// TIA Portal project "projeto_Grafcet" (V17)

(* hardware
DEVICE "S7-1500/ET200MP station_1"  S7-1500 station
   slot 0: "Rail_0"  Rack  6ES7 590-1***0-0AA0
   slot 1: "PLC_1"  CPU 1513-1 PN  6ES7 513-1AL02-0AB0  V2.9
      slot 3: "CPU display_1"  6ES7591-1AA00-0AA0
      slot 32768: "PROFINET interface_1"  X1
         slot 32769: "Port_1"  X1 P1
         slot 32770: "Port_2"  X1 P2
      slot 34817: "Virtual CP interface port_1"  Virtual CP interface port  Virtual CP interface port
   slot 2: "DI 32x24VDC SNK/SRC / DQ 32x24VDC/0.3A SNK BA_1"  DI 32x24VDC SNK/SRC / DQ 32x24VDC/0.3A SNK BA  6ES7 523-1BP50-0AA0  V1.0
*)

// ===== PLC "PLC_1"  CPU 1513-1 PN =====

VAR_GLOBAL   // PLC tag table "Default tag table"
   "Tag_3" AT %M2.2 : Bool;
   "Tag_4" AT %M2.0 : Bool;
   "Tag_1" AT %M2.4 : Bool;
   "Tag_5" AT %M2.5 : Bool;
   "Tag_2" AT %M3.3 : Bool;
   "Tag_6" AT %M3.4 : Bool;
   "Tag_7" AT %M2.6 : Bool;
   "Tag_8" AT %M2.7 : Bool;
   "Tag_9" AT %M3.0 : Bool;
   "Tag_10" AT %M3.1 : Bool;
   "M_1" AT %M1.3 : Bool;
   "M_2" AT %M1.4 : Bool;
   "MSaida" AT %M1.5 : Bool;
   "Limite Verde" AT %M1.6 : Bool;
   "MSAidaA" AT %M1.7 : Bool;
   "limite Azul" AT %M3.2 : Bool;
   "Mconta1" AT %M3.5 : Bool;
   "Mconta2" AT %M3.6 : Bool;
   "Terminou robo2" AT %M3.7 : Bool;
   "FACTORY I/O(Running)" AT %I1.7 : Bool;
   "Memo1" AT %M0.0 : Bool;
   "memo2" AT %M0.1 : Bool;
   "memo3" AT %M0.2 : Bool;
   "memo4" AT %M0.3 : Bool;
   "memo5" AT %M0.4 : Bool;
   "M_R2_Segura" AT %M0.5 : Bool;
   "M_R1_Segura" AT %M0.6 : Bool;
   "Limite_Ordenação" AT %M0.7 : Bool;
   "Sensor_borda_N" AT %M1.0 : Bool;
   "Fim_Etapa_Distribuição" AT %M1.1 : Bool;
   "termina_Distribuição" AT %M1.2 : Bool;
END_VAR

VAR_GLOBAL   // PLC tag table "Tag table_1"
   "R1 Sensor de Detecção de Peça" AT %I0.0 : Bool;
   "R2 Sensor de Detecção de Peça" AT %I0.1 : Bool;
   "R1 Sensor de Movimento Descer/Subir" AT %I0.2 : Bool;
   "R2 Sensor de Movimento Descer/Subir" AT %I0.3 : Bool;
   "R1 Sensor de Movimento Avançar/Recuar" AT %I0.4 : Bool;
   "R2 Sensor de Movimento Avançar/Recuar" AT %I0.5 : Bool;
   "Sensor de Saída 1" AT %I0.6 : Bool;
   "Sensor de Saída 2" AT %I0.7 : Bool;
   "Sensor do Organizador" AT %I1.0 : Bool;
   "Sensor Entrada Azul" AT %I1.1 : Bool;
   "Sensor Entrada Verde" AT %I1.2 : Bool;
   "Sensor Peça Azul" AT %I1.3 : Bool;
   "Sensor Peça Verde" AT %I1.4 : Bool;
   "Sensor Saída Azul" AT %I1.5 : Bool;
   "Sensor Saída Verde" AT %I1.6 : Bool;
   "Barreira" AT %Q0.0 : Bool;
   "Cinta do Desviador" AT %Q0.1 : Bool;
   "Deslocar Direita" AT %Q0.2 : Bool;
   "Deslocar Esquerda" AT %Q0.3 : Bool;
   "Desviador" AT %Q0.4 : Bool;
   "Esteira de Alimentação" AT %Q0.5 : Bool;
   "Esteira de Descarte P1" AT %Q0.6 : Bool;
   "Esteira de Descarte P2" AT %Q0.7 : Bool;
   "Esteira de Saída P1" AT %Q1.0 : Bool;
   "Esteira de Saída P2" AT %Q1.1 : Bool;
   "Esteira do Organizador" AT %Q1.2 : Bool;
   "Esteira Peça Azul  P1" AT %Q1.3 : Bool;
   "Esteira Peça Azul P2" AT %Q1.4 : Bool;
   "Esteira Peça Verde P1" AT %Q1.5 : Bool;
   "Esteira Peça Verde P2" AT %Q1.6 : Bool;
   "Esteira Peça Verde P3" AT %Q1.7 : Bool;
   "Esteira Peça Verde P4" AT %Q2.0 : Bool;
   "Esteira Peça Verde P5" AT %Q2.1 : Bool;
   "R1 Descer=1/Subir=0" AT %Q2.2 : Bool;
   "R2 Descer=1/Subir=0" AT %Q2.3 : Bool;
   "R1 Avançar=1/Recuar=0" AT %Q2.4 : Bool;
   "R1 Segurar=1/Soltar=0" AT %Q2.5 : Bool;
   "R2 Avançar=1/Recuar=0" AT %Q2.6 : Bool;
   "R2 Segurar=1/Soltar=0" AT %Q2.7 : Bool;
   "Receber Peça" AT %Q3.0 : Bool;
END_VAR

DATA_BLOCK "Separação_DB"   // DB6
{ S7_Optimized_Access := 'TRUE' }
VERSION : 0.1
// stored: InstanceOfName Separação
"Separação"
BEGIN
END_DATA_BLOCK

DATA_BLOCK "Block_1_DB"   // DB7
{ S7_Optimized_Access := 'TRUE' }
VERSION : 0.1
// stored: InstanceOfName Descarte
"Descarte"
BEGIN
END_DATA_BLOCK

DATA_BLOCK "Robo 2_DB"   // DB8
{ S7_Optimized_Access := 'TRUE' }
VERSION : 0.1
// stored: InstanceOfName Robo 2
"Robo 2"
BEGIN
END_DATA_BLOCK

DATA_BLOCK "Robo 1_DB"   // DB9
{ S7_Optimized_Access := 'TRUE' }
VERSION : 0.1
// stored: InstanceOfName Robo 1
"Robo 1"
BEGIN
END_DATA_BLOCK

DATA_BLOCK "Distribuição_DB"   // DB13
{ S7_Optimized_Access := 'TRUE' }
VERSION : 0.1
// stored: InstanceOfName Distribuição
"Distribuição"
BEGIN
END_DATA_BLOCK

// folder: System blocks/Program resources

DATA_BLOCK "IEC_Timer_0_DB"   // DB1
{ S7_Optimized_Access := 'TRUE' }
AUTHOR : Simatic
FAMILY : IEC
NAME : IEC_TMR
VERSION : 1.0
// stored: InstanceOfName IEC_TIMER
"IEC_TIMER"
BEGIN
END_DATA_BLOCK

DATA_BLOCK "IEC_Timer_0_DB_1"   // DB2
{ S7_Optimized_Access := 'TRUE' }
AUTHOR : Simatic
FAMILY : IEC
NAME : IEC_TMR
VERSION : 1.0
// stored: InstanceOfName IEC_TIMER
"IEC_TIMER"
BEGIN
END_DATA_BLOCK

DATA_BLOCK "IEC_Timer_0_DB_2"   // DB3
{ S7_Optimized_Access := 'TRUE' }
AUTHOR : Simatic
FAMILY : IEC
NAME : IEC_TMR
VERSION : 1.0
// stored: InstanceOfName IEC_TIMER
"IEC_TIMER"
BEGIN
END_DATA_BLOCK

DATA_BLOCK "IEC_Counter_0_DB"   // DB4
{ S7_Optimized_Access := 'TRUE' }
AUTHOR : Simatic
FAMILY : IEC
NAME : CNTR
VERSION : 1.0
// stored: InstanceOfName IEC_COUNTER
"IEC_COUNTER"
BEGIN
END_DATA_BLOCK

DATA_BLOCK "IEC_Counter_0_DB_1"   // DB5
{ S7_Optimized_Access := 'TRUE' }
AUTHOR : Simatic
FAMILY : IEC
NAME : CNTR
VERSION : 1.0
// stored: InstanceOfName IEC_COUNTER
"IEC_COUNTER"
BEGIN
END_DATA_BLOCK

DATA_BLOCK "IEC_Timer_0_DB_3"   // DB10
{ S7_Optimized_Access := 'TRUE' }
AUTHOR : Simatic
FAMILY : IEC
NAME : IEC_TMR
VERSION : 1.0
// stored: InstanceOfName IEC_TIMER
"IEC_TIMER"
BEGIN
END_DATA_BLOCK

DATA_BLOCK "IEC_Counter_0_DB_2"   // DB11
{ S7_Optimized_Access := 'TRUE' }
AUTHOR : Simatic
FAMILY : IEC
NAME : CNTR
VERSION : 1.0
// stored: InstanceOfName IEC_COUNTER
"IEC_COUNTER"
BEGIN
END_DATA_BLOCK

DATA_BLOCK "IEC_Counter_0_DB_3"   // DB12
{ S7_Optimized_Access := 'TRUE' }
AUTHOR : Simatic
FAMILY : IEC
NAME : CNTR
VERSION : 1.0
// stored: InstanceOfName IEC_COUNTER
"IEC_COUNTER"
BEGIN
END_DATA_BLOCK

// folder: (top level)

FUNCTION_BLOCK "Descarte"   // FB1, GRAPH_PLUS
{ S7_Optimized_Access := 'TRUE' }
VERSION : 0.1
   VAR_INPUT
      OFF_SQ : Bool := false;   // Turn sequence off
      INIT_SQ : Bool := false;   // Set sequence to initial state
      ACK_EF : Bool := false;   // Acknowledge all errors and faults
      S_PREV : Bool := false;   // Output previous step in parameter S_NO
      "Peça green" : Bool;
      S_NEXT : Bool := false;   // Indicate next step in parameter S_NO
      "peça blue" : Bool;
      SW_AUTO : Bool := false;   // Automatic mode
      SW_TAP : Bool := false;   // Semiautomatic/switch with transition
      SW_TOP : Bool := false;   // Semiautomatic/ignore transition
      SW_MAN : Bool := false;   // Manual mode
      S_SEL : Int := 0;   // Select step to be output to S_NO
      S_ON : Bool := false;   // Activate step indicated in S_NO
      S_OFF : Bool := false;   // Deactivate step indicated S_NO
      T_PUSH : Bool := false;   // Enable transition to switch in semi automatic mode
   END_VAR
   VAR_OUTPUT
      S_NO : Int := 0;   // Step number
      S_MORE : Bool := false;   // More steps are available and can be shown in S_NO
      S_ACTIVE : Bool := false;   // Step indicated in S_NO is active
      Cinta : Bool;
      ERR_FLT : Bool := false;   // Interlock or supervision group error
      AUTO_ON : Bool := false;   // Automatic mode is active
      D2 : Bool;
      D1 : Bool;
      Desviar_peça : Bool;
      TAP_ON : Bool := false;   // Semiautomatic mode/step with transition enabled
      TOP_ON : Bool := false;   // Semiautomatic mode/ignore transition enabled
      MAN_ON : Bool := false;   // Manual mode is active
   END_VAR
   VAR
      HMI_INFO : Array[0..8] of UInt;
      IF_PAR : G7_IfParPlus_V6;
      RT_DATA : G7_RTDataPlus_V6;   // Internal data area
      Trans3 : G7_TransitionPlus_V6;   // Transition structure
      Trans4 : G7_TransitionPlus_V6;   // Transition structure
      Trans5 : G7_TransitionPlus_V6;   // Transition structure
      Trans6 : G7_TransitionPlus_V6;   // Transition structure
      Step1 : G7_StepPlus_V6;   // Step structure
      Step2 : G7_StepPlus_V6;   // Step structure
      Step3 : G7_StepPlus_V6;   // Step structure
      Step4 : G7_StepPlus_V6;   // Step structure
      SINI : Array[0..1] of USInt;
      LSTT : Array[0..3] of USInt;
      ATAJ : Array[0..3] of USInt;
      ATAB : Array[0..3] of USInt;
      PSTT : Array[0..3] of USInt;
      NSTT : Array[0..3] of USInt;
      ASSJ : Array[0..3] of USInt;
      ASSB : Array[0..3] of USInt;
      PTTS : Array[0..3] of USInt;
      NTTS : Array[0..3] of USInt;
      SW_SQTS : Array[0..3] of USInt;
      SWITCH : Array[0..0] of USInt;
      TVX : Array[0..1] of USInt;
      TTX : Array[0..1] of USInt;
      TSX : Array[0..1] of USInt;
      S00X : Array[0..1] of USInt;
      SOFFX : Array[0..1] of USInt;
      SONX : Array[0..1] of USInt;
      SAX : Array[0..1] of USInt;
      SERRX : Array[0..4] of USInt;
      SMX : Array[0..4] of USInt;
      S0X : Array[0..4] of USInt;
      S1X : Array[0..4] of USInt;
      IL_ALARM_INST : Diag_Alarm;
      SUP_ALARM_INST : Diag_Alarm;
      STEP_TIME_ALARM_INST : Diag_Alarm;
      IEC_TIMER_INST : IEC_TIMER;
      TRANSACTION_FLAG : Bool := false;
   END_VAR
   // SINI[0] := 2;
   // PTTS[0] := 255;
   // TVX[0] := 16#1;
   // TTX[0] := 16#1;
   // TSX[0] := 16#1;
   // S00X[0] := 16#1;
   // SOFFX[0] := 16#1;
   // SONX[0] := 16#1;
   // SAX[0] := 16#1;
   // SERRX[0] := 16#1;
   // SMX[0] := 16#1;
   // S0X[0] := 16#1;
   // S1X[0] := 16#1;
   // LSTT[1] := 255;
   // ATAJ[1] := 1;
   // ATAJ[2] := 2;
   // ATAB[1] := 1;
   // ATAB[2] := 2;
   // PSTT[2] := 2;
   // NSTT[1] := 2;
   // ASSJ[1] := 1;
   // ASSB[1] := 1;
   // PTTS[2] := 1;
   // NTTS[2] := 2;
   // NTTS[1] := 1;
   // LSTT[0] := 255;
   // NSTT[0] := 1;
   // LSTT[2] := 255;
   // ATAJ[3] := 3;
   // ATAB[3] := 3;
   // PSTT[1] := 1;
   // PSTT[3] := 3;
   // NSTT[2] := 3;
   // ASSJ[2] := 2;
   // ASSJ[3] := 3;
   // ASSB[2] := 2;
   // ASSB[3] := 3;
   // PTTS[3] := 2;
   // NTTS[3] := 3;
BEGIN
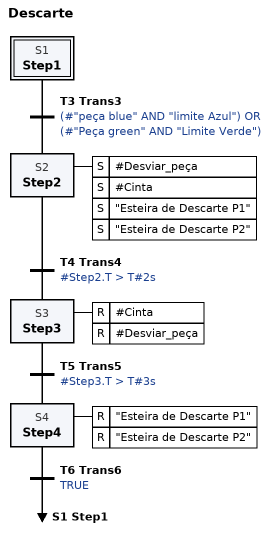
   // sequencer 1
   INITIAL_STEP Step1:   // S1, max time T#10S, warning time T#7S
   END_STEP
   TRANSITION Trans3 FROM Step1 TO Step2   // T3
      := (#"peça blue" AND "limite Azul") OR (#"Peça green" AND "Limite Verde");
   END_TRANSITION
   STEP Step2:   // S2, max time T#10S, warning time T#7S
              S    #Desviar_peça
              S    #Cinta
              S    "Esteira de Descarte P1"
              S    "Esteira de Descarte P2"
   END_STEP
   TRANSITION Trans4 FROM Step2 TO Step3   // T4
      := #Step2.T > T#2s;
   END_TRANSITION
   STEP Step3:   // S3, max time T#10S, warning time T#7S
              R    #Cinta
              R    #Desviar_peça
   END_STEP
   TRANSITION Trans5 FROM Step3 TO Step4   // T5
      := #Step3.T > T#3s;
   END_TRANSITION
   STEP Step4:   // S4, max time T#10S, warning time T#7S
              R    "Esteira de Descarte P1"
              R    "Esteira de Descarte P2"
   END_STEP
   TRANSITION Trans6 FROM Step4 TO Step1   // T6, jump
      := TRUE;
   END_TRANSITION
END_FUNCTION_BLOCK

FUNCTION_BLOCK "Separação"   // FB2, LAD
{ S7_Optimized_Access := 'TRUE' }
VERSION : 0.1
   VAR_INPUT
      "Sensor P verde" : Bool;
      "Sensor P azul" : Bool;
      "Sensor E azul" : Bool;
      "Sensor E Verde" : Bool;
      "Sensor S verde" : Bool;
      "Sensor S azul" : Bool;
      "Botao Start" : Bool;
   END_VAR
   VAR_OUTPUT
      "Est A P1" : Bool;
      "Est A P2" : Bool;
      "Deslocar Esquerda" : Bool;
      "Deslocar Direita" : Bool;
      "Receber Peça" : Bool;
      "Est Verde P1" : Bool;
      "Est Verde P2" : Bool;
      "Est Verde P3" : Bool;
      "Est Verde P4" : Bool;
      "Est Verde P5" : Bool;
   END_VAR
   VAR
      E1 : Bool;
      E2 : Bool;
      E3 : Bool;
      E4 : Bool;
      E5 : Bool;
      E6 : Bool;
      E7 : Bool;
      E8 : Bool;
      E9 : Bool;
      E10 : Bool;
      E11 : Bool;
      E12 : Bool;
   END_VAR
   VAR_TEMP   // added for the SCL form of the ladder/FBD networks
      _w1 : Bool;
      _w2 : Bool;
   END_VAR
BEGIN

REGION Network 1
   // Inicio do processo para o verde
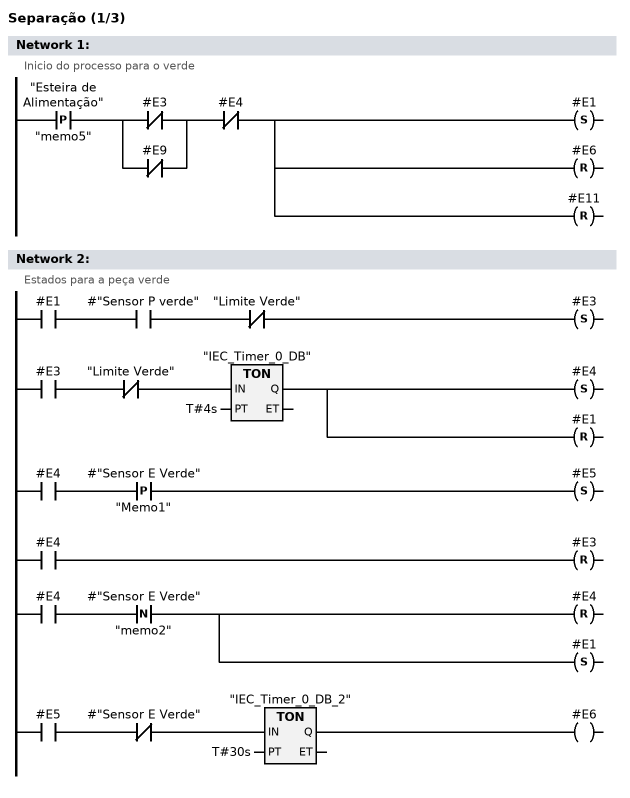
   RUNG wire#powerrail
      P_Contact(operand := "Esteira de Alimentação", bit := "memo5")
      wire#w1
      I_Contact( #E3 )
      wire#w2
      I_Contact( #E4 )
      wire#w3
      S_Coil( #E1 )
   END_RUNG
   RUNG wire#w1
      I_Contact( #E9 )
   END_RUNG wire#w2
   RUNG wire#w3
      R_Coil( #E6 )
   END_RUNG
   RUNG wire#w3
      R_Coil( #E11 )
   END_RUNG
   // the same network as SCL:
   #_w1 := "Esteira de Alimentação" AND NOT "memo5";   // rising edge of "Esteira de Alimentação"
   "memo5" := "Esteira de Alimentação";
   IF #_w1 AND (NOT #E3 OR NOT #E9) AND NOT #E4 THEN
       #E1 := TRUE;
       #E6 := FALSE;
       #E11 := FALSE;
   END_IF;
END_REGION

REGION Network 2
   // Estados para a peça verde
   IF #E1 AND #"Sensor P verde" AND NOT "Limite Verde" THEN #E3 := TRUE; END_IF;
   "IEC_Timer_0_DB".TON(IN := #E3 AND NOT "Limite Verde", PT := T#4s);
   IF "IEC_Timer_0_DB".Q THEN
       #E4 := TRUE;
       #E1 := FALSE;
   END_IF;
   #_w1 := #E4 AND #"Sensor E Verde" AND NOT "Memo1";   // rising edge of #"Sensor E Verde"
   "Memo1" := #"Sensor E Verde";
   IF #_w1 THEN #E5 := TRUE; END_IF;
   IF #E4 THEN #E3 := FALSE; END_IF;
   #_w2 := #E4 AND NOT #"Sensor E Verde" AND "memo2";   // falling edge of #"Sensor E Verde"
   "memo2" := #"Sensor E Verde";
   IF #_w2 THEN
       #E4 := FALSE;
       #E1 := TRUE;
   END_IF;
   "IEC_Timer_0_DB_2".TON(IN := #E5 AND NOT #"Sensor E Verde", PT := T#30s);
   #E6 := "IEC_Timer_0_DB_2".Q;
END_REGION

REGION Network 3
   // ações pro verde
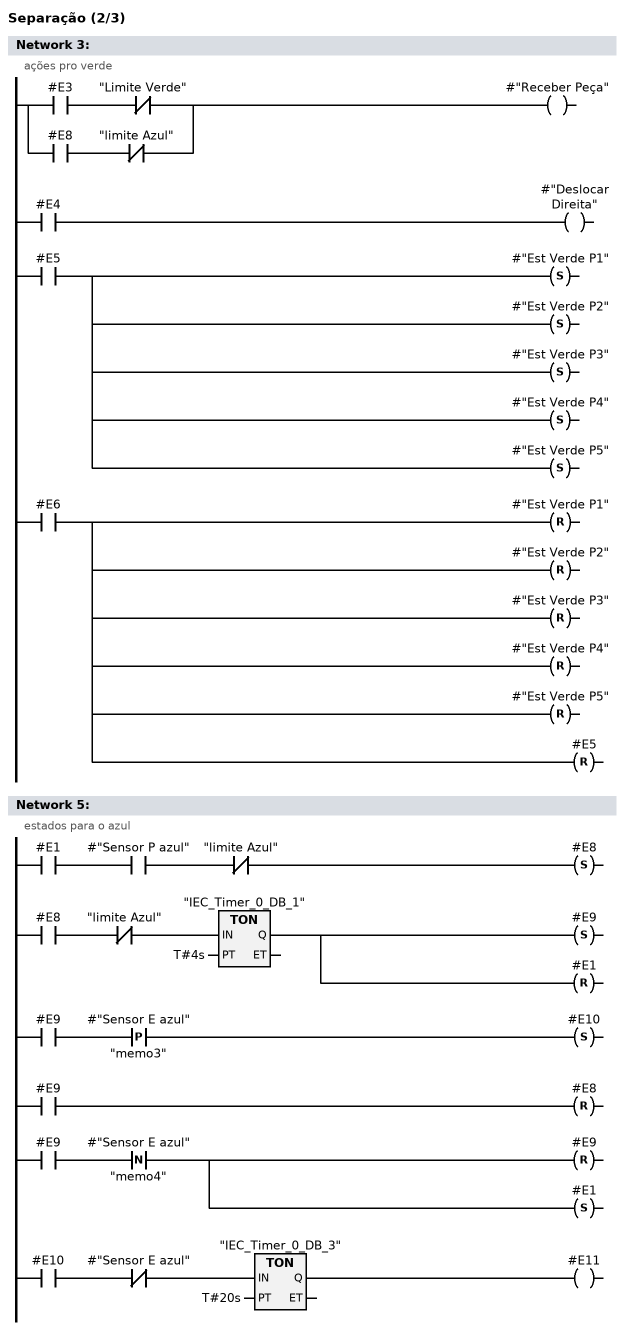
   RUNG wire#powerrail
      Contact( #E3 )
      I_Contact( "Limite Verde" )
      wire#w1
      Coil( #"Receber Peça" )
   END_RUNG
   RUNG wire#powerrail
      Contact( #E8 )
      I_Contact( "limite Azul" )
   END_RUNG wire#w1
   RUNG wire#powerrail
      Contact( #E4 )
      Coil( #"Deslocar Direita" )
   END_RUNG
   RUNG wire#powerrail
      Contact( #E5 )
      wire#w2
      S_Coil( #"Est Verde P1" )
   END_RUNG
   RUNG wire#w2
      S_Coil( #"Est Verde P2" )
   END_RUNG
   RUNG wire#w2
      S_Coil( #"Est Verde P3" )
   END_RUNG
   RUNG wire#w2
      S_Coil( #"Est Verde P4" )
   END_RUNG
   RUNG wire#w2
      S_Coil( #"Est Verde P5" )
   END_RUNG
   RUNG wire#powerrail
      Contact( #E6 )
      wire#w3
      R_Coil( #"Est Verde P1" )
   END_RUNG
   RUNG wire#w3
      R_Coil( #"Est Verde P2" )
   END_RUNG
   RUNG wire#w3
      R_Coil( #"Est Verde P3" )
   END_RUNG
   RUNG wire#w3
      R_Coil( #"Est Verde P4" )
   END_RUNG
   RUNG wire#w3
      R_Coil( #"Est Verde P5" )
   END_RUNG
   RUNG wire#w3
      R_Coil( #E5 )
   END_RUNG
   // the same network as SCL:
   #"Receber Peça" := (#E3 AND NOT "Limite Verde") OR (#E8 AND NOT "limite Azul");
   #"Deslocar Direita" := #E4;
   IF #E5 THEN
       #"Est Verde P1" := TRUE;
       #"Est Verde P2" := TRUE;
       #"Est Verde P3" := TRUE;
       #"Est Verde P4" := TRUE;
       #"Est Verde P5" := TRUE;
   END_IF;
   IF #E6 THEN
       #"Est Verde P1" := FALSE;
       #"Est Verde P2" := FALSE;
       #"Est Verde P3" := FALSE;
       #"Est Verde P4" := FALSE;
       #"Est Verde P5" := FALSE;
       #E5 := FALSE;
   END_IF;
END_REGION

REGION Network 4
   // inicio para o azul
END_REGION

REGION Network 5
   // estados para o azul
   IF #E1 AND #"Sensor P azul" AND NOT "limite Azul" THEN #E8 := TRUE; END_IF;
   "IEC_Timer_0_DB_1".TON(IN := #E8 AND NOT "limite Azul", PT := T#4s);
   IF "IEC_Timer_0_DB_1".Q THEN
       #E9 := TRUE;
       #E1 := FALSE;
   END_IF;
   #_w1 := #E9 AND #"Sensor E azul" AND NOT "memo3";   // rising edge of #"Sensor E azul"
   "memo3" := #"Sensor E azul";
   IF #_w1 THEN #E10 := TRUE; END_IF;
   IF #E9 THEN #E8 := FALSE; END_IF;
   #_w2 := #E9 AND NOT #"Sensor E azul" AND "memo4";   // falling edge of #"Sensor E azul"
   "memo4" := #"Sensor E azul";
   IF #_w2 THEN
       #E9 := FALSE;
       #E1 := TRUE;
   END_IF;
   "IEC_Timer_0_DB_3".TON(IN := #E10 AND NOT #"Sensor E azul", PT := T#20s);
   #E11 := "IEC_Timer_0_DB_3".Q;
END_REGION

REGION Network 6
   // ações pra peça azul
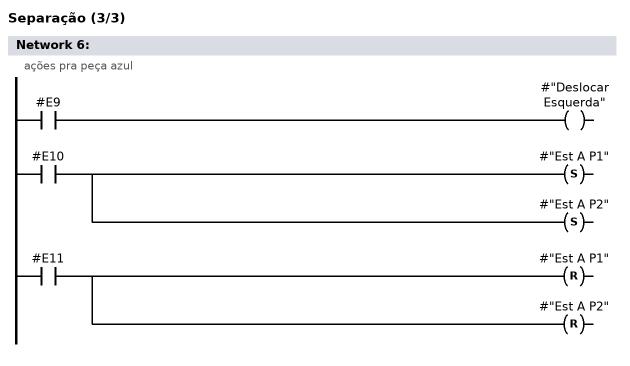
   RUNG wire#powerrail
      Contact( #E9 )
      Coil( #"Deslocar Esquerda" )
   END_RUNG
   RUNG wire#powerrail
      Contact( #E10 )
      wire#w1
      S_Coil( #"Est A P1" )
   END_RUNG
   RUNG wire#w1
      S_Coil( #"Est A P2" )
   END_RUNG
   RUNG wire#powerrail
      Contact( #E11 )
      wire#w2
      R_Coil( #"Est A P1" )
   END_RUNG
   RUNG wire#w2
      R_Coil( #"Est A P2" )
   END_RUNG
   // the same network as SCL:
   #"Deslocar Esquerda" := #E9;
   IF #E10 THEN
       #"Est A P1" := TRUE;
       #"Est A P2" := TRUE;
   END_IF;
   IF #E11 THEN
       #"Est A P1" := FALSE;
       #"Est A P2" := FALSE;
   END_IF;
END_REGION
END_FUNCTION_BLOCK

FUNCTION_BLOCK "Robo 2"   // FB3, GRAPH_PLUS
{ S7_Optimized_Access := 'TRUE' }
VERSION : 0.1
   VAR_INPUT
      OFF_SQ : Bool := false;   // Turn sequence off
      INIT_SQ : Bool := false;   // Set sequence to initial state
      Sensor_saida_green : Bool;
      ACK_EF : Bool := false;   // Acknowledge all errors and faults
      "Sensor Avança" : Bool;
      "Sensor Detecção de peça" : Bool;
      S_PREV : Bool := false;   // Output previous step in parameter S_NO
      "Sensor descer" : Bool;
      S_NEXT : Bool := false;   // Indicate next step in parameter S_NO
      SW_AUTO : Bool := false;   // Automatic mode
      SW_TAP : Bool := false;   // Semiautomatic/switch with transition
      SW_TOP : Bool := false;   // Semiautomatic/ignore transition
      SW_MAN : Bool := false;   // Manual mode
      S_SEL : Int := 0;   // Select step to be output to S_NO
      S_ON : Bool := false;   // Activate step indicated in S_NO
      S_OFF : Bool := false;   // Deactivate step indicated S_NO
      T_PUSH : Bool := false;   // Enable transition to switch in semi automatic mode
   END_VAR
   VAR_OUTPUT
      S_NO : Int := 0;   // Step number
      S_MORE : Bool := false;   // More steps are available and can be shown in S_NO
      "Agarrar peça" : Bool;
      Avançar : Bool;
      Output_1 : Bool;
      S_ACTIVE : Bool := false;   // Step indicated in S_NO is active
      Descer : Bool;
      ERR_FLT : Bool := false;   // Interlock or supervision group error
      AUTO_ON : Bool := false;   // Automatic mode is active
      TAP_ON : Bool := false;   // Semiautomatic mode/step with transition enabled
      TOP_ON : Bool := false;   // Semiautomatic mode/ignore transition enabled
      MAN_ON : Bool := false;   // Manual mode is active
   END_VAR
   VAR
      HMI_INFO : Array[0..8] of UInt;
      IF_PAR : G7_IfParPlus_V6;
      RT_DATA : G7_RTDataPlus_V6;   // Internal data area
      Trans1 : G7_TransitionPlus_V6;   // Transition structure
      Trans2 : G7_TransitionPlus_V6;   // Transition structure
      Trans3 : G7_TransitionPlus_V6;   // Transition structure
      Trans4 : G7_TransitionPlus_V6;   // Transition structure
      Trans5 : G7_TransitionPlus_V6;   // Transition structure
      Trans6 : G7_TransitionPlus_V6;   // Transition structure
      Trans7 : G7_TransitionPlus_V6;   // Transition structure
      Trans8 : G7_TransitionPlus_V6;   // Transition structure
      Trans9 : G7_TransitionPlus_V6;   // Transition structure
      Step1 : G7_StepPlus_V6;   // Step structure
      Step2 : G7_StepPlus_V6;   // Step structure
      Step3 : G7_StepPlus_V6;   // Step structure
      Step4 : G7_StepPlus_V6;   // Step structure
      Step5 : G7_StepPlus_V6;   // Step structure
      Step6 : G7_StepPlus_V6;   // Step structure
      Step7 : G7_StepPlus_V6;   // Step structure
      Step8 : G7_StepPlus_V6;   // Step structure
      Step9 : G7_StepPlus_V6;   // Step structure
      SINI : Array[0..1] of USInt;
      LSTT : Array[0..8] of USInt;
      ATAJ : Array[0..8] of USInt;
      ATAB : Array[0..8] of USInt;
      PSTT : Array[0..8] of USInt;
      NSTT : Array[0..8] of USInt;
      ASSJ : Array[0..8] of USInt;
      ASSB : Array[0..8] of USInt;
      PTTS : Array[0..8] of USInt;
      NTTS : Array[0..8] of USInt;
      SW_SQTS : Array[0..8] of USInt;
      SWITCH : Array[0..0] of USInt;
      TVX : Array[0..1] of USInt;
      TTX : Array[0..1] of USInt;
      TSX : Array[0..1] of USInt;
      S00X : Array[0..1] of USInt;
      SOFFX : Array[0..1] of USInt;
      SONX : Array[0..1] of USInt;
      SAX : Array[0..1] of USInt;
      SERRX : Array[0..9] of USInt;
      SMX : Array[0..9] of USInt;
      S0X : Array[0..9] of USInt;
      S1X : Array[0..9] of USInt;
      IL_ALARM_INST : Diag_Alarm;
      SUP_ALARM_INST : Diag_Alarm;
      STEP_TIME_ALARM_INST : Diag_Alarm;
      IEC_TIMER_INST : IEC_TIMER;
      TRANSACTION_FLAG : Bool := false;
   END_VAR
   // SINI[0] := 2;
   // LSTT[0] := 255;
   // LSTT[1] := 255;
   // LSTT[2] := 255;
   // LSTT[3] := 255;
   // LSTT[4] := 255;
   // LSTT[5] := 255;
   // LSTT[6] := 255;
   // LSTT[7] := 255;
   // ATAJ[1] := 1;
   // ATAJ[2] := 2;
   // ATAJ[3] := 3;
   // ATAJ[4] := 4;
   // ATAJ[5] := 5;
   // ATAJ[6] := 6;
   // ATAJ[7] := 7;
   // ATAJ[8] := 8;
   // ATAB[1] := 1;
   // ATAB[2] := 2;
   // ATAB[3] := 3;
   // ATAB[4] := 4;
   // ATAB[5] := 5;
   // ATAB[6] := 6;
   // ATAB[7] := 7;
   // ATAB[8] := 8;
   // PSTT[1] := 1;
   // PSTT[2] := 2;
   // PSTT[3] := 3;
   // PSTT[4] := 4;
   // PSTT[5] := 5;
   // PSTT[6] := 6;
   // PSTT[7] := 7;
   // PSTT[8] := 8;
   // NSTT[0] := 1;
   // NSTT[1] := 2;
   // NSTT[2] := 3;
   // NSTT[3] := 4;
   // NSTT[4] := 5;
   // NSTT[5] := 6;
   // NSTT[6] := 7;
   // NSTT[7] := 8;
   // ASSJ[1] := 1;
   // ASSJ[2] := 2;
   // ASSJ[3] := 3;
   // ASSJ[4] := 4;
   // ASSJ[5] := 5;
   // ASSJ[6] := 6;
   // ASSJ[7] := 7;
   // ASSJ[8] := 8;
   // ASSB[1] := 1;
   // ASSB[2] := 2;
   // ASSB[3] := 3;
   // ASSB[4] := 4;
   // ASSB[5] := 5;
   // ASSB[6] := 6;
   // ASSB[7] := 7;
   // ASSB[8] := 8;
   // PTTS[0] := 255;
   // PTTS[2] := 1;
   // PTTS[3] := 2;
   // PTTS[4] := 3;
   // PTTS[5] := 4;
   // PTTS[6] := 5;
   // PTTS[7] := 6;
   // PTTS[8] := 7;
   // NTTS[1] := 1;
   // NTTS[2] := 2;
   // NTTS[3] := 3;
   // NTTS[4] := 4;
   // NTTS[5] := 5;
   // NTTS[6] := 6;
   // NTTS[7] := 7;
   // NTTS[8] := 8;
   // TVX[0] := 16#1;
   // TTX[0] := 16#1;
   // TSX[0] := 16#1;
   // S00X[0] := 16#1;
   // SOFFX[0] := 16#1;
   // SONX[0] := 16#1;
   // SAX[0] := 16#1;
   // SERRX[0] := 16#1;
   // SMX[0] := 16#1;
   // S0X[0] := 16#1;
   // S1X[0] := 16#1;
BEGIN
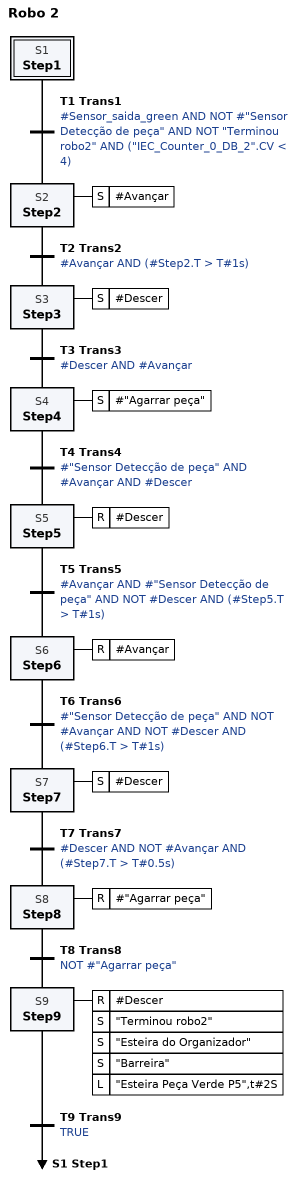
   // sequencer 1
   INITIAL_STEP Step1:   // S1, max time T#10S, warning time T#7S
   END_STEP
   TRANSITION Trans1 FROM Step1 TO Step2   // T1
      := #Sensor_saida_green AND NOT #"Sensor Detecção de peça" AND NOT "Terminou robo2" AND ("IEC_Counter_0_DB_2".CV < 4);
   END_TRANSITION
   STEP Step2:   // S2, max time T#10S, warning time T#7S
              S    #Avançar
   END_STEP
   TRANSITION Trans2 FROM Step2 TO Step3   // T2
      := #Avançar AND (#Step2.T > T#1s);
   END_TRANSITION
   STEP Step3:   // S3, max time T#10S, warning time T#7S
              S    #Descer
   END_STEP
   TRANSITION Trans3 FROM Step3 TO Step4   // T3
      := #Descer AND #Avançar;
   END_TRANSITION
   STEP Step4:   // S4, max time T#10S, warning time T#7S
              S    #"Agarrar peça"
   END_STEP
   TRANSITION Trans4 FROM Step4 TO Step5   // T4
      := #"Sensor Detecção de peça" AND #Avançar AND #Descer;
   END_TRANSITION
   STEP Step5:   // S5, max time T#10S, warning time T#7S
              R    #Descer
   END_STEP
   TRANSITION Trans5 FROM Step5 TO Step6   // T5
      := #Avançar AND #"Sensor Detecção de peça" AND NOT #Descer AND (#Step5.T > T#1s);
   END_TRANSITION
   STEP Step6:   // S6, max time T#10S, warning time T#7S
              R    #Avançar
   END_STEP
   TRANSITION Trans6 FROM Step6 TO Step7   // T6
      := #"Sensor Detecção de peça" AND NOT #Avançar AND NOT #Descer AND (#Step6.T > T#1s);
   END_TRANSITION
   STEP Step7:   // S7, max time T#10S, warning time T#7S
              S    #Descer
   END_STEP
   TRANSITION Trans7 FROM Step7 TO Step8   // T7
      := #Descer AND NOT #Avançar AND (#Step7.T > T#0.5s);
   END_TRANSITION
   STEP Step8:   // S8, max time T#10S, warning time T#7S
              R    #"Agarrar peça"
   END_STEP
   TRANSITION Trans8 FROM Step8 TO Step9   // T8
      := NOT #"Agarrar peça";
   END_TRANSITION
   STEP Step9:   // S9, max time T#10S, warning time T#7S
              R    #Descer
              S    "Terminou robo2"
              S    "Esteira do Organizador"
              S    "Barreira"
              L    "Esteira Peça Verde P5",t#2S
   END_STEP
   TRANSITION Trans9 FROM Step9 TO Step1   // T9, jump
      := TRUE;
   END_TRANSITION
END_FUNCTION_BLOCK

FUNCTION_BLOCK "Robo 1"   // FB4, GRAPH_PLUS
{ S7_Optimized_Access := 'TRUE' }
VERSION : 0.1
   VAR_INPUT
      "Sensor descer" : Bool;
      "Sensor detecção de peça_1" : Bool;
      "Sensor Avança" : Bool;
      "Terminou R2" : Bool;
      "Sensor detecção de peça" : Bool;
      Saída_blue : Bool;
   END_VAR
   VAR_OUTPUT
      "agarrar peça" : Bool;
      descer : Bool;
      avançar : Bool;
   END_VAR
   VAR
      HMI_INFO : Array[0..8] of UInt;
      IF_PAR : G7_IfParPlus_V6;
      RT_DATA : G7_RTDataPlus_V6;   // Internal data area
      Trans1 : G7_TransitionPlus_V6;   // Transition structure
      Trans2 : G7_TransitionPlus_V6;   // Transition structure
      Trans3 : G7_TransitionPlus_V6;   // Transition structure
      Trans4 : G7_TransitionPlus_V6;   // Transition structure
      Trans5 : G7_TransitionPlus_V6;   // Transition structure
      Trans6 : G7_TransitionPlus_V6;   // Transition structure
      Trans7 : G7_TransitionPlus_V6;   // Transition structure
      Trans8 : G7_TransitionPlus_V6;   // Transition structure
      Trans9 : G7_TransitionPlus_V6;   // Transition structure
      Step1 : G7_StepPlus_V6;   // Step structure
      Step2 : G7_StepPlus_V6;   // Step structure
      Step3 : G7_StepPlus_V6;   // Step structure
      Step4 : G7_StepPlus_V6;   // Step structure
      Step5 : G7_StepPlus_V6;   // Step structure
      Step6 : G7_StepPlus_V6;   // Step structure
      Step7 : G7_StepPlus_V6;   // Step structure
      Step8 : G7_StepPlus_V6;   // Step structure
      Step9 : G7_StepPlus_V6;   // Step structure
      SINI : Array[0..1] of USInt;
      LSTT : Array[0..8] of USInt;
      ATAJ : Array[0..8] of USInt;
      ATAB : Array[0..8] of USInt;
      PSTT : Array[0..8] of USInt;
      NSTT : Array[0..8] of USInt;
      ASSJ : Array[0..8] of USInt;
      ASSB : Array[0..8] of USInt;
      PTTS : Array[0..8] of USInt;
      NTTS : Array[0..8] of USInt;
      SW_SQTS : Array[0..8] of USInt;
      SWITCH : Array[0..0] of USInt;
      TVX : Array[0..1] of USInt;
      TTX : Array[0..1] of USInt;
      TSX : Array[0..1] of USInt;
      S00X : Array[0..1] of USInt;
      SOFFX : Array[0..1] of USInt;
      SONX : Array[0..1] of USInt;
      SAX : Array[0..1] of USInt;
      SERRX : Array[0..9] of USInt;
      SMX : Array[0..9] of USInt;
      S0X : Array[0..9] of USInt;
      S1X : Array[0..9] of USInt;
      IL_ALARM_INST : Diag_Alarm;
      SUP_ALARM_INST : Diag_Alarm;
      STEP_TIME_ALARM_INST : Diag_Alarm;
      IEC_TIMER_INST : IEC_TIMER;
      TRANSACTION_FLAG : Bool := false;
   END_VAR
   // SINI[0] := 2;
   // LSTT[0] := 255;
   // LSTT[1] := 255;
   // LSTT[2] := 255;
   // LSTT[3] := 255;
   // LSTT[4] := 255;
   // LSTT[5] := 255;
   // LSTT[6] := 255;
   // LSTT[7] := 255;
   // ATAJ[1] := 1;
   // ATAJ[2] := 2;
   // ATAJ[3] := 3;
   // ATAJ[4] := 4;
   // ATAJ[5] := 5;
   // ATAJ[6] := 6;
   // ATAJ[7] := 7;
   // ATAJ[8] := 8;
   // ATAB[1] := 1;
   // ATAB[2] := 2;
   // ATAB[3] := 3;
   // ATAB[4] := 4;
   // ATAB[5] := 5;
   // ATAB[6] := 6;
   // ATAB[7] := 7;
   // ATAB[8] := 8;
   // PSTT[1] := 1;
   // PSTT[2] := 2;
   // PSTT[3] := 3;
   // PSTT[4] := 4;
   // PSTT[5] := 5;
   // PSTT[6] := 6;
   // PSTT[7] := 7;
   // PSTT[8] := 8;
   // NSTT[0] := 1;
   // NSTT[1] := 2;
   // NSTT[2] := 3;
   // NSTT[3] := 4;
   // NSTT[4] := 5;
   // NSTT[5] := 6;
   // NSTT[6] := 7;
   // NSTT[7] := 8;
   // ASSJ[1] := 1;
   // ASSJ[2] := 2;
   // ASSJ[3] := 3;
   // ASSJ[4] := 4;
   // ASSJ[5] := 5;
   // ASSJ[6] := 6;
   // ASSJ[7] := 7;
   // ASSJ[8] := 8;
   // ASSB[1] := 1;
   // ASSB[2] := 2;
   // ASSB[3] := 3;
   // ASSB[4] := 4;
   // ASSB[5] := 5;
   // ASSB[6] := 6;
   // ASSB[7] := 7;
   // ASSB[8] := 8;
   // PTTS[0] := 255;
   // PTTS[2] := 1;
   // PTTS[3] := 2;
   // PTTS[4] := 3;
   // PTTS[5] := 4;
   // PTTS[6] := 5;
   // PTTS[7] := 6;
   // PTTS[8] := 7;
   // NTTS[1] := 1;
   // NTTS[2] := 2;
   // NTTS[3] := 3;
   // NTTS[4] := 4;
   // NTTS[5] := 5;
   // NTTS[6] := 6;
   // NTTS[7] := 7;
   // NTTS[8] := 8;
   // TVX[0] := 16#1;
   // TTX[0] := 16#1;
   // TSX[0] := 16#1;
   // S00X[0] := 16#1;
   // SOFFX[0] := 16#1;
   // SONX[0] := 16#1;
   // SAX[0] := 16#1;
   // SERRX[0] := 16#1;
   // SMX[0] := 16#1;
   // S0X[0] := 16#1;
   // S1X[0] := 16#1;
BEGIN
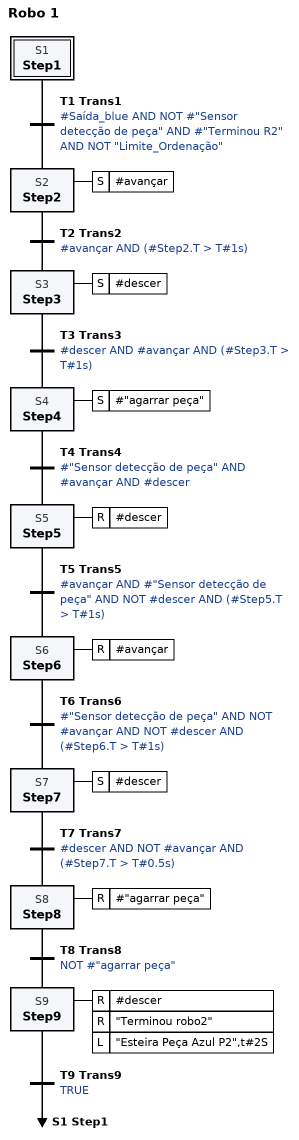
   // sequencer 1
   INITIAL_STEP Step1:   // S1, max time T#10S, warning time T#7S
   END_STEP
   TRANSITION Trans1 FROM Step1 TO Step2   // T1
      := #Saída_blue AND NOT #"Sensor detecção de peça" AND #"Terminou R2" AND NOT "Limite_Ordenação";
   END_TRANSITION
   STEP Step2:   // S2, max time T#10S, warning time T#7S
              S    #avançar
   END_STEP
   TRANSITION Trans2 FROM Step2 TO Step3   // T2
      := #avançar AND (#Step2.T > T#1s);
   END_TRANSITION
   STEP Step3:   // S3, max time T#10S, warning time T#7S
              S    #descer
   END_STEP
   TRANSITION Trans3 FROM Step3 TO Step4   // T3
      := #descer AND #avançar AND (#Step3.T > T#1s);
   END_TRANSITION
   STEP Step4:   // S4, max time T#10S, warning time T#7S
              S    #"agarrar peça"
   END_STEP
   TRANSITION Trans4 FROM Step4 TO Step5   // T4
      := #"Sensor detecção de peça" AND #avançar AND #descer;
   END_TRANSITION
   STEP Step5:   // S5, max time T#10S, warning time T#7S
              R    #descer
   END_STEP
   TRANSITION Trans5 FROM Step5 TO Step6   // T5
      := #avançar AND #"Sensor detecção de peça" AND NOT #descer AND (#Step5.T > T#1s);
   END_TRANSITION
   STEP Step6:   // S6, max time T#10S, warning time T#7S
              R    #avançar
   END_STEP
   TRANSITION Trans6 FROM Step6 TO Step7   // T6
      := #"Sensor detecção de peça" AND NOT #avançar AND NOT #descer AND (#Step6.T > T#1s);
   END_TRANSITION
   STEP Step7:   // S7, max time T#10S, warning time T#7S
              S    #descer
   END_STEP
   TRANSITION Trans7 FROM Step7 TO Step8   // T7
      := #descer AND NOT #avançar AND (#Step7.T > T#0.5s);
   END_TRANSITION
   STEP Step8:   // S8, max time T#10S, warning time T#7S
              R    #"agarrar peça"
   END_STEP
   TRANSITION Trans8 FROM Step8 TO Step9   // T8
      := NOT #"agarrar peça";
   END_TRANSITION
   STEP Step9:   // S9, max time T#10S, warning time T#7S
              R    #descer
              R    "Terminou robo2"
              L    "Esteira Peça Azul P2",t#2S
   END_STEP
   TRANSITION Trans9 FROM Step9 TO Step1   // T9, jump
      := TRUE;
   END_TRANSITION
END_FUNCTION_BLOCK

FUNCTION_BLOCK "Distribuição"   // FB5, GRAPH_PLUS
{ S7_Optimized_Access := 'TRUE' }
VERSION : 0.1
   VAR
      HMI_INFO : Array[0..8] of UInt;
      IF_PAR : G7_IfParPlus_V6;
      RT_DATA : G7_RTDataPlus_V6;   // Internal data area
      Trans1 : G7_TransitionPlus_V6;   // Transition structure
      Trans2 : G7_TransitionPlus_V6;   // Transition structure
      Trans3 : G7_TransitionPlus_V6;   // Transition structure
      Trans4 : G7_TransitionPlus_V6;   // Transition structure
      Trans5 : G7_TransitionPlus_V6;   // Transition structure
      Trans6 : G7_TransitionPlus_V6;   // Transition structure
      Trans7 : G7_TransitionPlus_V6;   // Transition structure
      Trans8 : G7_TransitionPlus_V6;   // Transition structure
      Trans9 : G7_TransitionPlus_V6;   // Transition structure
      Step1 : G7_StepPlus_V6;   // Step structure
      Step2 : G7_StepPlus_V6;   // Step structure
      Step3 : G7_StepPlus_V6;   // Step structure
      Step4 : G7_StepPlus_V6;   // Step structure
      Step5 : G7_StepPlus_V6;   // Step structure
      Step6 : G7_StepPlus_V6;   // Step structure
      Step7 : G7_StepPlus_V6;   // Step structure
      Step8 : G7_StepPlus_V6;   // Step structure
      SINI : Array[0..1] of USInt;
      LSTT : Array[0..8] of USInt;
      ATAJ : Array[0..8] of USInt;
      ATAB : Array[0..8] of USInt;
      PSTT : Array[0..8] of USInt;
      NSTT : Array[0..8] of USInt;
      ASSJ : Array[0..7] of USInt;
      ASSB : Array[0..7] of USInt;
      PTTS : Array[0..7] of USInt;
      NTTS : Array[0..7] of USInt;
      SW_SQTS : Array[0..7] of USInt;
      SWITCH : Array[0..0] of USInt;
      TVX : Array[0..3] of USInt;
      TTX : Array[0..3] of USInt;
      TSX : Array[0..1] of USInt;
      S00X : Array[0..1] of USInt;
      SOFFX : Array[0..1] of USInt;
      SONX : Array[0..1] of USInt;
      SAX : Array[0..1] of USInt;
      SERRX : Array[0..8] of USInt;
      SMX : Array[0..8] of USInt;
      S0X : Array[0..8] of USInt;
      S1X : Array[0..8] of USInt;
      IL_ALARM_INST : Diag_Alarm;
      SUP_ALARM_INST : Diag_Alarm;
      STEP_TIME_ALARM_INST : Diag_Alarm;
      IEC_TIMER_INST : IEC_TIMER;
      TRANSACTION_FLAG : Bool := false;
   END_VAR
   // SINI[0] := 2;
   // LSTT[0] := 255;
   // LSTT[1] := 255;
   // LSTT[2] := 255;
   // LSTT[3] := 255;
   // LSTT[4] := 255;
   // LSTT[6] := 1;
   // ATAJ[1] := 1;
   // ATAJ[2] := 2;
   // ATAJ[3] := 3;
   // ATAJ[4] := 4;
   // ATAJ[5] := 5;
   // ATAJ[6] := 6;
   // ATAB[1] := 1;
   // ATAB[2] := 2;
   // ATAB[3] := 3;
   // ATAB[4] := 4;
   // ATAB[5] := 6;
   // ATAB[6] := 5;
   // PSTT[1] := 1;
   // PSTT[2] := 2;
   // PSTT[3] := 3;
   // PSTT[4] := 4;
   // PSTT[5] := 5;
   // PSTT[6] := 5;
   // NSTT[0] := 1;
   // NSTT[1] := 2;
   // NSTT[2] := 3;
   // NSTT[3] := 4;
   // NSTT[4] := 5;
   // NSTT[6] := 1;
   // ASSJ[1] := 1;
   // ASSJ[2] := 2;
   // ASSJ[3] := 3;
   // ASSJ[4] := 4;
   // ASSJ[5] := 5;
   // ASSB[1] := 1;
   // ASSB[2] := 2;
   // ASSB[3] := 3;
   // ASSB[4] := 4;
   // ASSB[5] := 5;
   // PTTS[0] := 255;
   // PTTS[2] := 1;
   // PTTS[3] := 2;
   // PTTS[4] := 3;
   // PTTS[5] := 4;
   // NTTS[1] := 1;
   // NTTS[2] := 2;
   // NTTS[3] := 3;
   // NTTS[4] := 4;
   // NTTS[5] := 5;
   // TVX[0] := 16#1;
   // TTX[0] := 16#1;
   // TSX[0] := 16#1;
   // S00X[0] := 16#1;
   // SOFFX[0] := 16#1;
   // SONX[0] := 16#1;
   // SAX[0] := 16#1;
   // SERRX[0] := 16#1;
   // SMX[0] := 16#1;
   // S0X[0] := 16#1;
   // S1X[0] := 16#1;
   // ATAJ[8] := 8;
   // ATAJ[7] := 7;
   // LSTT[7] := 255;
   // LSTT[5] := 255;
   // ATAB[7] := 7;
   // ATAB[8] := 8;
   // PSTT[7] := 6;
   // PSTT[8] := 7;
   // NSTT[5] := 6;
   // NSTT[7] := 7;
   // ASSJ[6] := 6;
   // ASSJ[7] := 7;
   // ASSB[6] := 6;
   // ASSB[7] := 7;
   // PTTS[6] := 5;
   // PTTS[7] := 7;
   // NTTS[6] := 7;
   // NTTS[7] := 8;
   // SW_SQTS[6] := 1;
   // SW_SQTS[7] := 1;
BEGIN
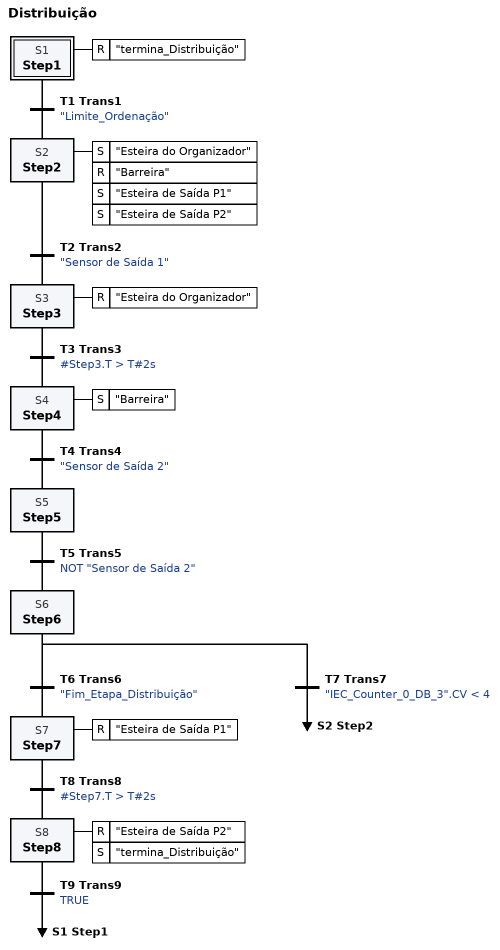
   // sequencer 1
   INITIAL_STEP Step1:   // S1, max time T#10S, warning time T#7S
              R    "termina_Distribuição"
   END_STEP
   TRANSITION Trans1 FROM Step1 TO Step2   // T1
      := "Limite_Ordenação";
   END_TRANSITION
   STEP Step2:   // S2, max time T#10S, warning time T#7S
              S    "Esteira do Organizador"
              R    "Barreira"
              S    "Esteira de Saída P1"
              S    "Esteira de Saída P2"
   END_STEP
   TRANSITION Trans2 FROM Step2 TO Step3   // T2
      := "Sensor de Saída 1";
   END_TRANSITION
   STEP Step3:   // S3, max time T#10S, warning time T#7S
              R    "Esteira do Organizador"
   END_STEP
   TRANSITION Trans3 FROM Step3 TO Step4   // T3
      := #Step3.T > T#2s;
   END_TRANSITION
   STEP Step4:   // S4, max time T#10S, warning time T#7S
              S    "Barreira"
   END_STEP
   TRANSITION Trans4 FROM Step4 TO Step5   // T4
      := "Sensor de Saída 2";
   END_TRANSITION
   STEP Step5:   // S5, max time T#10S, warning time T#7S
   END_STEP
   TRANSITION Trans5 FROM Step5 TO Step6   // T5
      := NOT "Sensor de Saída 2";
   END_TRANSITION
   STEP Step6:   // S6, max time T#10S, warning time T#7S
   END_STEP
   TRANSITION Trans6 FROM Step6 TO Step7   // T6
      := "Fim_Etapa_Distribuição";
   END_TRANSITION
   TRANSITION Trans7 FROM Step6 TO Step2   // T7, jump
      := "IEC_Counter_0_DB_3".CV < 4;
   END_TRANSITION
   STEP Step7:   // S7, max time T#10S, warning time T#7S
              R    "Esteira de Saída P1"
   END_STEP
   TRANSITION Trans8 FROM Step7 TO Step8   // T8
      := #Step7.T > T#2s;
   END_TRANSITION
   STEP Step8:   // S8, max time T#10S, warning time T#7S
              R    "Esteira de Saída P2"
              S    "termina_Distribuição"
   END_STEP
   TRANSITION Trans9 FROM Step8 TO Step1   // T9, jump
      := TRUE;
   END_TRANSITION
END_FUNCTION_BLOCK

ORGANIZATION_BLOCK "Main"   // OB1, LAD, ProgramCycle
TITLE = "Main Program Sweep (Cycle)"
{ S7_Optimized_Access := 'TRUE' }
VERSION : 0.1
   VAR_INPUT
      Initial_Call : Bool;   // Initial call of this OB
      Remanence : Bool;   // =True, if remanent data are available
   END_VAR
   VAR_TEMP   // added for the SCL form of the ladder/FBD networks
      _w1 : Bool;
      _w2 : Bool;
   END_VAR
BEGIN

REGION Network 1
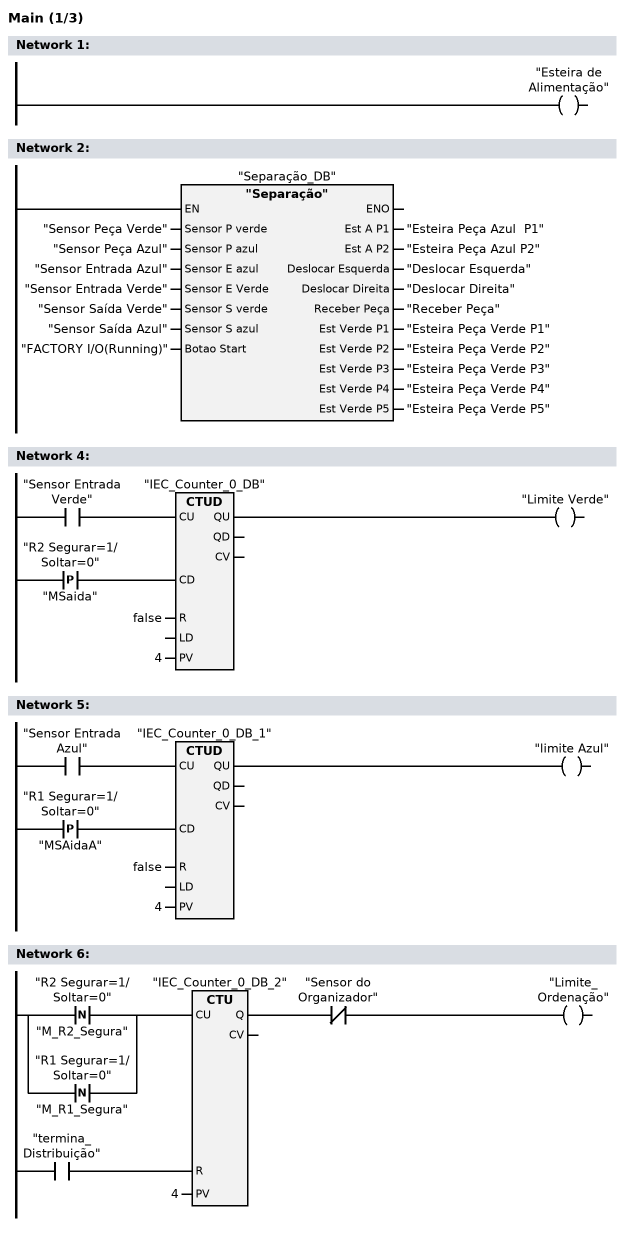
   RUNG wire#powerrail
      Coil( "Esteira de Alimentação" )
   END_RUNG
   // the same network as SCL:
   "Esteira de Alimentação" := TRUE;
END_REGION

REGION Network 2
   RUNG wire#powerrail
      "Separação_DB"("Sensor P verde" := "Sensor Peça Verde", "Sensor P azul" := "Sensor Peça Azul", "Sensor E azul" := "Sensor Entrada Azul", "Sensor E Verde" := "Sensor Entrada Verde", "Sensor S verde" := "Sensor Saída Verde", "Sensor S azul" := "Sensor Saída Azul", "Botao Start" := "FACTORY I/O(Running)", "Est A P1" => "Esteira Peça Azul  P1", "Est A P2" => "Esteira Peça Azul P2", "Deslocar Esquerda" => "Deslocar Esquerda", "Deslocar Direita" => "Deslocar Direita", "Receber Peça" => "Receber Peça", "Est Verde P1" => "Esteira Peça Verde P1", "Est Verde P2" => "Esteira Peça Verde P2", "Est Verde P3" => "Esteira Peça Verde P3", "Est Verde P4" => "Esteira Peça Verde P4", "Est Verde P5" => "Esteira Peça Verde P5")
   END_RUNG
   // the same network as SCL:
   "Separação_DB"("Sensor P verde" := "Sensor Peça Verde",   // "Separação"
                  "Sensor P azul" := "Sensor Peça Azul",
                  "Sensor E azul" := "Sensor Entrada Azul",
                  "Sensor E Verde" := "Sensor Entrada Verde",
                  "Sensor S verde" := "Sensor Saída Verde",
                  "Sensor S azul" := "Sensor Saída Azul",
                  "Botao Start" := "FACTORY I/O(Running)",
                  "Est A P1" => "Esteira Peça Azul  P1",
                  "Est A P2" => "Esteira Peça Azul P2",
                  "Deslocar Esquerda" => "Deslocar Esquerda",
                  "Deslocar Direita" => "Deslocar Direita",
                  "Receber Peça" => "Receber Peça",
                  "Est Verde P1" => "Esteira Peça Verde P1",
                  "Est Verde P2" => "Esteira Peça Verde P2",
                  "Est Verde P3" => "Esteira Peça Verde P3",
                  "Est Verde P4" => "Esteira Peça Verde P4",
                  "Est Verde P5" => "Esteira Peça Verde P5");
END_REGION

REGION Network 4
   #_w1 := "R2 Segurar=1/Soltar=0" AND NOT "MSaida";   // rising edge of "R2 Segurar=1/Soltar=0"
   "MSaida" := "R2 Segurar=1/Soltar=0";
   "IEC_Counter_0_DB".CTUD(CU := "Sensor Entrada Verde", CD := #_w1, R := false, PV := 4);
   "Limite Verde" := "IEC_Counter_0_DB".QU;
END_REGION

REGION Network 5
   #_w1 := "R1 Segurar=1/Soltar=0" AND NOT "MSAidaA";   // rising edge of "R1 Segurar=1/Soltar=0"
   "MSAidaA" := "R1 Segurar=1/Soltar=0";
   "IEC_Counter_0_DB_1".CTUD(CU := "Sensor Entrada Azul", CD := #_w1, R := false, PV := 4);
   "limite Azul" := "IEC_Counter_0_DB_1".QU;
END_REGION

REGION Network 6
   #_w1 := NOT "R2 Segurar=1/Soltar=0" AND "M_R2_Segura";   // falling edge of "R2 Segurar=1/Soltar=0"
   "M_R2_Segura" := "R2 Segurar=1/Soltar=0";
   #_w2 := NOT "R1 Segurar=1/Soltar=0" AND "M_R1_Segura";   // falling edge of "R1 Segurar=1/Soltar=0"
   "M_R1_Segura" := "R1 Segurar=1/Soltar=0";
   "IEC_Counter_0_DB_2".CTU(CU := #_w1 OR #_w2, R := "termina_Distribuição", PV := 4);
   "Limite_Ordenação" := "IEC_Counter_0_DB_2".Q AND NOT "Sensor do Organizador";
END_REGION

REGION Network 7
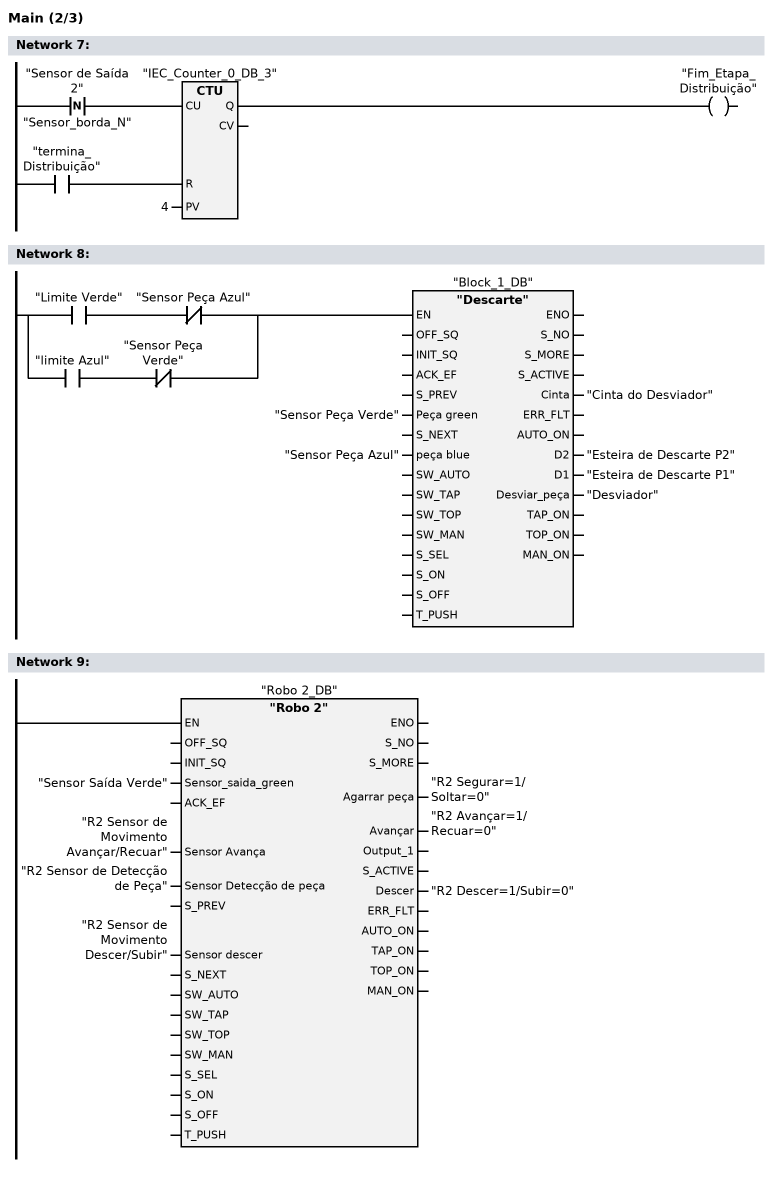
   #_w1 := NOT "Sensor de Saída 2" AND "Sensor_borda_N";   // falling edge of "Sensor de Saída 2"
   "Sensor_borda_N" := "Sensor de Saída 2";
   "IEC_Counter_0_DB_3".CTU(CU := #_w1, R := "termina_Distribuição", PV := 4);
   "Fim_Etapa_Distribuição" := "IEC_Counter_0_DB_3".Q;
END_REGION

REGION Network 8
   RUNG wire#powerrail
      Contact( "Limite Verde" )
      I_Contact( "Sensor Peça Azul" )
      wire#w1
      "Block_1_DB"(OFF_SQ :=, INIT_SQ :=, ACK_EF :=, S_PREV :=, "Peça green" := "Sensor Peça Verde", S_NEXT :=, "peça blue" := "Sensor Peça Azul", SW_AUTO :=, SW_TAP :=, SW_TOP :=, SW_MAN :=, S_SEL :=, S_ON :=, S_OFF :=, T_PUSH :=, S_NO =>, S_MORE =>, S_ACTIVE =>, Cinta => "Cinta do Desviador", ERR_FLT =>, AUTO_ON =>, D2 => "Esteira de Descarte P2", D1 => "Esteira de Descarte P1", Desviar_peça => "Desviador", TAP_ON =>, TOP_ON =>, MAN_ON =>)
   END_RUNG
   RUNG wire#powerrail
      Contact( "limite Azul" )
      I_Contact( "Sensor Peça Verde" )
   END_RUNG wire#w1
   // the same network as SCL:
   IF ("Limite Verde" AND NOT "Sensor Peça Azul") OR ("limite Azul" AND NOT "Sensor Peça Verde") THEN
       "Block_1_DB"("Peça green" := "Sensor Peça Verde",   // "Descarte"
                    "peça blue" := "Sensor Peça Azul",
                    Cinta => "Cinta do Desviador",
                    D2 => "Esteira de Descarte P2",
                    D1 => "Esteira de Descarte P1",
                    Desviar_peça => "Desviador");
   END_IF;
END_REGION

REGION Network 9
   RUNG wire#powerrail
      "Robo 2_DB"(OFF_SQ :=, INIT_SQ :=, Sensor_saida_green := "Sensor Saída Verde", ACK_EF :=, "Sensor Avança" := "R2 Sensor de Movimento Avançar/Recuar", "Sensor Detecção de peça" := "R2 Sensor de Detecção de Peça", S_PREV :=, "Sensor descer" := "R2 Sensor de Movimento Descer/Subir", S_NEXT :=, SW_AUTO :=, SW_TAP :=, SW_TOP :=, SW_MAN :=, S_SEL :=, S_ON :=, S_OFF :=, T_PUSH :=, S_NO =>, S_MORE =>, "Agarrar peça" => "R2 Segurar=1/Soltar=0", Avançar => "R2 Avançar=1/Recuar=0", Output_1 =>, S_ACTIVE =>, Descer => "R2 Descer=1/Subir=0", ERR_FLT =>, AUTO_ON =>, TAP_ON =>, TOP_ON =>, MAN_ON =>)
   END_RUNG
   // the same network as SCL:
   "Robo 2_DB"(Sensor_saida_green := "Sensor Saída Verde",   // "Robo 2"
               "Sensor Avança" := "R2 Sensor de Movimento Avançar/Recuar",
               "Sensor Detecção de peça" := "R2 Sensor de Detecção de Peça",
               "Sensor descer" := "R2 Sensor de Movimento Descer/Subir",
               "Agarrar peça" => "R2 Segurar=1/Soltar=0",
               Avançar => "R2 Avançar=1/Recuar=0",
               Descer => "R2 Descer=1/Subir=0");
END_REGION

REGION Network 10
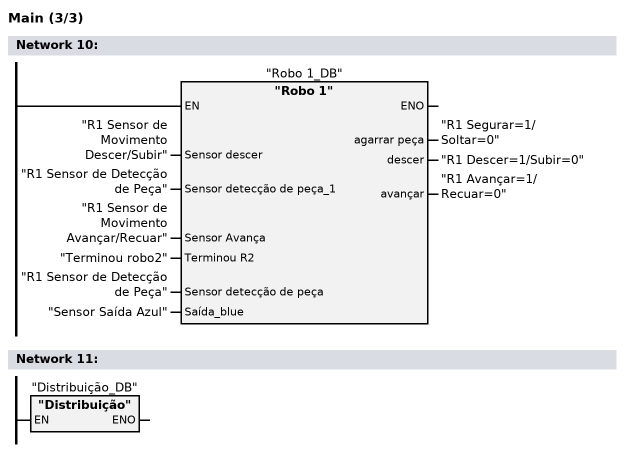
   RUNG wire#powerrail
      "Robo 1_DB"("Sensor descer" := "R1 Sensor de Movimento Descer/Subir", "Sensor detecção de peça_1" := "R1 Sensor de Detecção de Peça", "Sensor Avança" := "R1 Sensor de Movimento Avançar/Recuar", "Terminou R2" := "Terminou robo2", "Sensor detecção de peça" := "R1 Sensor de Detecção de Peça", Saída_blue := "Sensor Saída Azul", "agarrar peça" => "R1 Segurar=1/Soltar=0", descer => "R1 Descer=1/Subir=0", avançar => "R1 Avançar=1/Recuar=0")
   END_RUNG
   // the same network as SCL:
   "Robo 1_DB"("Sensor descer" := "R1 Sensor de Movimento Descer/Subir",   // "Robo 1"
               "Sensor detecção de peça_1" := "R1 Sensor de Detecção de Peça",
               "Sensor Avança" := "R1 Sensor de Movimento Avançar/Recuar",
               "Terminou R2" := "Terminou robo2",
               "Sensor detecção de peça" := "R1 Sensor de Detecção de Peça",
               Saída_blue := "Sensor Saída Azul",
               "agarrar peça" => "R1 Segurar=1/Soltar=0",
               descer => "R1 Descer=1/Subir=0",
               avançar => "R1 Avançar=1/Recuar=0");
END_REGION

REGION Network 11
   RUNG wire#powerrail
      "Distribuição_DB"()
   END_RUNG
   // the same network as SCL:
   "Distribuição_DB"();   // "Distribuição"
END_REGION
END_ORGANIZATION_BLOCK